SREFP 3 C00063 BC00063  +REFP EC00063
CALL JOB:SEARCH-R1-S13D
SET P054 P006
SFTON3D P054
SMOVL C00064 BC00064 V=166.7  +MOVJ EC00064
SMOVL C00065 BC00065 V=416.7  +MOVJ EC00065
SMOVL C00066 BC00066 V=250.0  +MOVJ EC00066
SREFP 3 C00067 BC00067  +REFP EC00067
CALL JOB:SEARCH-R1-S13D
SET P054 P006
SFTON3D P054
SMOVL C00068 BC00068 V=250.0  +MOVJ EC00068
MOVL C00069 BC00069 V=1000.0  +MOVJ EC00069 VJ=100.00
'EndPath S4207
'Path S4095
SFTOF3D
MOVJ C00070 BC00070 VJ=100.00  +MOVJ EC00070 VJ=100.00
MOVJ C00071 BC00071 VJ=100.00  +MOVJ EC00071 VJ=100.00
SMOVL C00072 BC00072 V=200.0  +MOVJ EC00072
SREFP 3 C00073 BC00073  +REFP EC00073
CALL JOB:SEARCH-R1-S13D
SET P089 P006
SFTON3D P089
SMOVL C00074 BC00074 V=166.7  +MOVJ EC00074
SMOVL C00075 BC00075 V=166.7  +MOVJ EC00075
SREFP 3 C00076 BC00076  +REFP EC00076
CALL JOB:SEARCH-R1-S13D
SET P089 P006
SFTON3D P089
SMOVL C00077 BC00077 V=166.7  +MOVJ EC00077
SMOVL C00078 BC00078 V=166.7  +MOVJ EC00078
SREFP 3 C00079 BC00079  +REFP EC00079
CALL JOB:SEARCH-R1-S13D
SET P089 P006
SFTON3D P089
SMOVL C00080 BC00080 V=166.7  +MOVJ EC00080
SMOVL C00081 BC00081 V=1000.0  +MOVJ EC00081
SFTOF3D
MOVJ C00082 BC00082 VJ=100.00  +MOVJ EC00082 VJ=100.00
MOVL C00083 BC00083 V=666.7  +MOVJ EC00083 VJ=100.00
SMOVL C00084 BC00084 V=166.7  +MOVJ EC00084
SREFP 3 C00085 BC00085  +REFP EC00085
CALL JOB:SEARCH-R1-S13D
SET P034 P006
SFTON3D P034
SMOVL C00086 BC00086 V=250.0  +MOVJ EC00086
SMOVL C00087 BC00087 V=233.3  +MOVJ EC00087
SMOVL C00088 BC00088 V=166.7  +MOVJ EC00088
SREFP 3 C00089 BC00089  +REFP EC00089
CALL JOB:SEARCH-R1-S13D
SET P034 P006
SFTON3D P034
SMOVL C00090 BC00090 V=166.7  +MOVJ EC00090
SMOVL C00091 BC00091 V=166.7  +MOVJ EC00091
SREFP 3 C00092 BC00092  +REFP EC00092
CALL JOB:SEARCH-R1-S13D
SET P034 P006
SFTON3D P034
SMOVL C00093 BC00093 V=166.7  +MOVJ EC00093
MOVJ C00094 BC00094 VJ=50.00  +MOVJ EC00094 VJ=30.00
'EndPath S4095
'Path S4096
SFTOF3D
MOVJ C00095 BC00095 VJ=50.00  +MOVJ EC00095 VJ=30.00
MOVJ C00096 BC00096 VJ=50.00  +MOVJ EC00096 VJ=30.00
MOVJ C00097 BC00097 VJ=50.00  +MOVJ EC00097 VJ=30.00
SMOVL C00098 BC00098 V=166.7  +MOVJ EC00098
SREFP 3 C00099 BC00099  +REFP EC00099
CALL JOB:SEARCH-R1-S13D
SET P061 P006
SFTON3D P061
SMOVL C00100 BC00100 V=166.7  +MOVJ EC00100
SREFP 3 C00101 BC00101  +REFP EC00101
CALL JOB:SEARCH-R1-S13D
SET P061 P006
SFTON3D P061
SMOVL C00102 BC00102 V=166.7  +MOVJ EC00102
SFTOF3D
SMOVL C00103 BC00103 V=666.7  +MOVJ EC00103
SMOVL C00104 BC00104 V=166.7  +MOVJ EC00104
SREFP 3 C00105 BC00105  +REFP EC00105
CALL JOB:SEARCH-R1-S13D
SET P062 P006
SFTON3D P062
SMOVL C00106 BC00106 V=166.7  +MOVJ EC00106
SREFP 3 C00107 BC00107  +REFP EC00107
CALL JOB:SEARCH-R1-S13D
SET P062 P006
SFTON3D P062
SMOVL C00108 BC00108 V=250.0  +MOVJ EC00108
SFTOF3D
SMOVL C00109 BC00109 V=500.0  +MOVJ EC00109
SMOVL C00110 BC00110 V=166.7  +MOVJ EC00110
SREFP 3 C00111 BC00111  +REFP EC00111
CALL JOB:SEARCH-R1-S13D
SET P063 P006
SFTON3D P063
SMOVL C00112 BC00112 V=166.7  +MOVJ EC00112
SREFP 3 C00113 BC00113  +REFP EC00113
CALL JOB:SEARCH-R1-S13D
SET P063 P006
SFTON3D P063
SMOVL C00114 BC00114 V=166.7  +MOVJ EC00114
SFTOF3D
SMOVL C00115 BC00115 V=1000.0  +MOVJ EC00115
MOVJ C00116 BC00116 VJ=100.00  +MOVJ EC00116 VJ=30.00
MOVJ C00117 BC00117 VJ=50.00  +MOVJ EC00117 VJ=30.00
MOVJ C00118 BC00118 VJ=100.00  +MOVJ EC00118 VJ=100.00
MOVL C00119 BC00119 V=666.7  +MOVJ EC00119 VJ=100.00
SMOVL C00120 BC00120 V=166.7  +MOVJ EC00120
SREFP 3 C00121 BC00121  +REFP EC00121
CALL JOB:SEARCH-R1-S13D
SET P023 P006
SFTON3D P023
SMOVL C00122 BC00122 V=166.7  +MOVJ EC00122
SMOVL C00123 BC00123 V=333.3  +MOVJ EC00123
SMOVL C00124 BC00124 V=166.7  +MOVJ EC00124
SREFP 3 C00125 BC00125  +REFP EC00125
CALL JOB:SEARCH-R1-S13D
SET P023 P006
SFTON3D P023
SMOVL C00126 BC00126 V=166.7  +MOVJ EC00126
SMOVL C00127 BC00127 V=166.7  +MOVJ EC00127
SREFP 3 C00128 BC00128  +REFP EC00128
CALL JOB:SEARCH-R1-S13D
SET P023 P006
SFTON3D P023
SMOVL C00129 BC00129 V=166.7  +MOVJ EC00129
MOVL C00130 BC00130 V=1000.0  +MOVJ EC00130 VJ=100.00
'EndPath S4096
MOVJ C00131 BC00131 VJ=100.00  +MOVJ EC00131 VJ=100.00
'Path S4097
SFTOF3D
MOVJ C00132 BC00132 VJ=100.00  +MOVJ EC00132 VJ=100.00
MOVL C00133 BC00133 V=666.7  +MOVJ EC00133 VJ=100.00
SMOVL C00134 BC00134 V=166.7  +MOVJ EC00134
SREFP 3 C00135 BC00135  +REFP EC00135
CALL JOB:SEARCH-R1-S13D
SET P024 P006
SFTON3D P024
SMOVL C00136 BC00136 V=166.7  +MOVJ EC00136
SREFP 3 C00137 BC00137  +REFP EC00137
CALL JOB:SEARCH-R1-S13D
SET P024 P006
SFTON3D P024
SMOVL C00138 BC00138 V=166.7  +MOVJ EC00138
SMOVL C00139 BC00139 V=166.7  +MOVJ EC00139
SREFP 3 C00140 BC00140  +REFP EC00140
CALL JOB:SEARCH-R1-S13D
SET P024 P006
SFTON3D P024
SMOVL C00141 BC00141 V=166.7  +MOVJ EC00141
MOVL C00142 BC00142 V=1000.0  +MOVJ EC00142 VJ=100.00
'EndPath S4097
'Path S4098
SFTOF3D
MOVJ C00143 BC00143 VJ=100.00  +MOVJ EC00143 VJ=100.00
MOVL C00144 BC00144 V=666.7  +MOVJ EC00144 VJ=100.00
SMOVL C00145 BC00145 V=166.7  +MOVJ EC00145
SREFP 3 C00146 BC00146  +REFP EC00146
CALL JOB:SEARCH-R1-S13D
SET P035 P006
SFTON3D P035
SMOVL C00147 BC00147 V=166.7  +MOVJ EC00147
SREFP 3 C00148 BC00148  +REFP EC00148
CALL JOB:SEARCH-R1-S13D
SET P035 P006
SFTON3D P035
SMOVL C00149 BC00149 V=166.7  +MOVJ EC00149
SMOVL C00150 BC00150 V=166.7  +MOVJ EC00150
SMOVL C00151 BC00151 V=166.7  +MOVJ EC00151
SREFP 3 C00152 BC00152  +REFP EC00152
CALL JOB:SEARCH-R1-S13D
SET P035 P006
SFTON3D P035
SMOVL C00153 BC00153 V=166.7  +MOVJ EC00153
MOVL C00154 BC00154 V=1000.0  +MOVJ EC00154 VJ=100.00
'EndPath S4098
'Path S4099
SFTOF3D
MOVJ C00155 BC00155 VJ=100.00  +MOVJ EC00155 VJ=100.00
MOVL C00156 BC00156 V=666.7  +MOVJ EC00156 VJ=100.00
SMOVL C00157 BC00157 V=166.7  +MOVJ EC00157
SREFP 3 C00158 BC00158  +REFP EC00158
CALL JOB:SEARCH-R1-S13D
SET P029 P006
SFTON3D P029
SMOVL C00159 BC00159 V=166.7  +MOVJ EC00159
SREFP 3 C00160 BC00160  +REFP EC00160
CALL JOB:SEARCH-R1-S13D
SET P029 P006
SFTON3D P029
SMOVL C00161 BC00161 V=166.7  +MOVJ EC00161
SMOVL C00162 BC00162 V=250.0  +MOVJ EC00162
SMOVL C00163 BC00163 V=166.7  +MOVJ EC00163
SREFP 3 C00164 BC00164  +REFP EC00164
CALL JOB:SEARCH-R1-S13D
SET P029 P006
SFTON3D P029
SMOVL C00165 BC00165 V=166.7  +MOVJ EC00165
'EndPath S4099
'Path S4855
SFTOF3D
MOVL C00166 BC00166 V=666.7  +MOVJ EC00166 VJ=100.00
SMOVL C00167 BC00167 V=166.7  +MOVJ EC00167
SREFP 3 C00168 BC00168  +REFP EC00168
CALL JOB:SEARCH-R1-S13D
SET P071 P006
SFTON3D P071
SMOVL C00169 BC00169 V=166.7  +MOVJ EC00169
SREFP 3 C00170 BC00170  +REFP EC00170
CALL JOB:SEARCH-R1-S13D
SET P071 P006
SFTON3D P071
SMOVL C00171 BC00171 V=166.7  +MOVJ EC00171
SMOVL C00172 BC00172 V=166.7  +MOVJ EC00172
SREFP 3 C00173 BC00173  +REFP EC00173
CALL JOB:SEARCH-R1-S13D
SET P071 P006
SFTON3D P071
SMOVL C00174 BC00174 V=166.7  +MOVJ EC00174
MOVL C00175 BC00175 V=1000.0  +MOVJ EC00175 VJ=100.00
'EndPath S4855
'Path S4856
SFTOF3D
MOVJ C00176 BC00176 VJ=100.00  +MOVJ EC00176 VJ=100.00
MOVL C00177 BC00177 V=666.7  +MOVJ EC00177 VJ=100.00
SMOVL C00178 BC00178 V=166.7  +MOVJ EC00178
SREFP 3 C00179 BC00179  +REFP EC00179
CALL JOB:SEARCH-R1-S13D
SET P072 P006
SFTON3D P072
SMOVL C00180 BC00180 V=166.7  +MOVJ EC00180
SREFP 3 C00181 BC00181  +REFP EC00181
CALL JOB:SEARCH-R1-S13D
SET P072 P006
SFTON3D P072
SMOVL C00182 BC00182 V=166.7  +MOVJ EC00182
MOVL C00183 BC00183 V=1000.0  +MOVJ EC00183 VJ=100.00
'EndPath S4856
MOVJ C00184 BC00184 VJ=100.00  +MOVJ EC00184 VJ=100.00
'Path S4857
SFTOF3D
MOVJ C00185 BC00185 VJ=100.00  +MOVJ EC00185 VJ=100.00
MOVL C00186 BC00186 V=666.7  +MOVJ EC00186 VJ=100.00
SMOVL C00187 BC00187 V=166.7  +MOVJ EC00187
SREFP 3 C00188 BC00188  +REFP EC00188
CALL JOB:SEARCH-R1-S13D
SET P073 P006
SFTON3D P073
SMOVL C00189 BC00189 V=166.7  +MOVJ EC00189
SMOVL C00190 BC00190 V=166.7  +MOVJ EC00190
SREFP 3 C00191 BC00191  +REFP EC00191
CALL JOB:SEARCH-R1-S13D
SET P073 P006
SFTON3D P073
SMOVL C00192 BC00192 V=166.7  +MOVJ EC00192
SMOVL C00193 BC00193 V=166.7  +MOVJ EC00193
SREFP 3 C00194 BC00194  +REFP EC00194
CALL JOB:SEARCH-R1-S13D
SET P073 P006
SFTON3D P073
SMOVL C00195 BC00195 V=166.7  +MOVJ EC00195
MOVL C00196 BC00196 V=1000.0  +MOVJ EC00196 VJ=100.00
'EndPath S4857
MOVJ C00197 BC00197 VJ=100.00  +MOVJ EC00197 VJ=100.00
'Path S4858
SFTOF3D
MOVJ C00198 BC00198 VJ=100.00  +MOVJ EC00198 VJ=100.00
MOVL C00199 BC00199 V=666.7  +MOVJ EC00199 VJ=100.00
SMOVL C00200 BC00200 V=166.7  +MOVJ EC00200
SREFP 3 C00201 BC00201  +REFP EC00201
CALL JOB:SEARCH-R1-S13D
SET P074 P006
SFTON3D P074
SMOVL C00202 BC00202 V=166.7  +MOVJ EC00202
SREFP 3 C00203 BC00203  +REFP EC00203
CALL JOB:SEARCH-R1-S13D
SET P074 P006
SFTON3D P074
SMOVL C00204 BC00204 V=166.7  +MOVJ EC00204
MOVL C00205 BC00205 V=1000.0  +MOVJ EC00205 VJ=100.00
'EndPath S4858
MOVJ C00206 BC00206 VJ=100.00  +MOVJ EC00206 VJ=100.00
MOVJ C00207 BC00207 VJ=100.00  +MOVJ EC00207 VJ=100.00
'Path S4100
SFTOF3D
MOVJ C00208 BC00208 VJ=100.00  +MOVJ EC00208 VJ=100.00
MOVL C00209 BC00209 V=666.7  +MOVJ EC00209 VJ=100.00
SMOVL C00210 BC00210 V=166.7  +MOVJ EC00210
SREFP 3 C00211 BC00211  +REFP EC00211
CALL JOB:SEARCH-R1-S13D
SET P026 P006
SFTON3D P026
SMOVL C00212 BC00212 V=166.7  +MOVJ EC00212
SREFP 3 C00213 BC00213  +REFP EC00213
CALL JOB:SEARCH-R1-S13D
SET P026 P006
SFTON3D P026
SMOVL C00214 BC00214 V=166.7  +MOVJ EC00214
SMOVL C00215 BC00215 V=666.7  +MOVJ EC00215
SMOVL C00216 BC00216 V=666.7  +MOVJ EC00216
SMOVL C00217 BC00217 V=666.7  +MOVJ EC00217
SMOVL C00218 BC00218 V=166.7  +MOVJ EC00218
SREFP 3 C00219 BC00219  +REFP EC00219
CALL JOB:SEARCH-R1-S13D
SET P026 P006
SFTON3D P026
SMOVL C00220 BC00220 V=250.0  +MOVJ EC00220
SMOVL C00221 BC00221 V=666.7  +MOVJ EC00221
MOVL C00222 BC00222 V=1000.0  +MOVJ EC00222 VJ=100.00
'EndPath S4100
MOVJ C00223 BC00223 VJ=50.00  +MOVJ EC00223 VJ=100.00
'Path S4101
SFTOF3D
MOVJ C00224 BC00224 VJ=50.00  +MOVJ EC00224 VJ=100.00
MOVL C00225 BC00225 V=666.7  +MOVJ EC00225 VJ=100.00
SMOVL C00226 BC00226 V=166.7  +MOVJ EC00226
SREFP 3 C00227 BC00227  +REFP EC00227
CALL JOB:SEARCH-R1-S13D
SET P025 P006
SFTON3D P025
SMOVL C00228 BC00228 V=166.7  +MOVJ EC00228
SREFP 3 C00229 BC00229  +REFP EC00229
CALL JOB:SEARCH-R1-S13D
SET P025 P006
SFTON3D P025
SMOVL C00230 BC00230 V=166.7  +MOVJ EC00230
SMOVL C00231 BC00231 V=333.3  +MOVJ EC00231
SMOVL C00232 BC00232 V=166.7  +MOVJ EC00232
SREFP 3 C00233 BC00233  +REFP EC00233
CALL JOB:SEARCH-R1-S13D
SET P025 P006
SFTON3D P025
SMOVL C00234 BC00234 V=166.7  +MOVJ EC00234
MOVL C00235 BC00235 V=1000.0  +MOVJ EC00235 VJ=100.00
'EndPath S4101
MOVJ C00236 BC00236 VJ=100.00  +MOVJ EC00236 VJ=100.00
'Path S4102
SFTOF3D
MOVJ C00237 BC00237 VJ=100.00  +MOVJ EC00237 VJ=100.00
MOVL C00238 BC00238 V=666.7  +MOVJ EC00238 VJ=100.00
SMOVL C00239 BC00239 V=166.7  +MOVJ EC00239
SREFP 3 C00240 BC00240  +REFP EC00240
CALL JOB:SEARCH-R1-S13D
SET P028 P006
SFTON3D P028
SMOVL C00241 BC00241 V=166.7  +MOVJ EC00241
SREFP 3 C00242 BC00242  +REFP EC00242
CALL JOB:SEARCH-R1-S13D
SET P028 P006
SFTON3D P028
SMOVL C00243 BC00243 V=166.7  +MOVJ EC00243
SMOVL C00244 BC00244 V=333.3  +MOVJ EC00244
SMOVL C00245 BC00245 V=166.7  +MOVJ EC00245
SREFP 3 C00246 BC00246  +REFP EC00246
CALL JOB:SEARCH-R1-S13D
SET P028 P006
SFTON3D P028
SMOVL C00247 BC00247 V=166.7  +MOVJ EC00247
MOVL C00248 BC00248 V=1000.0  +MOVJ EC00248 VJ=100.00
'EndPath S4102
MOVJ C00249 BC00249 VJ=100.00  +MOVJ EC00249 VJ=100.00
'Path S4103
SFTOF3D
MOVJ C00250 BC00250 VJ=100.00  +MOVJ EC00250 VJ=100.00
MOVL C00251 BC00251 V=666.7  +MOVJ EC00251 VJ=100.00
SMOVL C00252 BC00252 V=166.7  +MOVJ EC00252
SREFP 3 C00253 BC00253  +REFP EC00253
CALL JOB:SEARCH-R1-S13D
SET P033 P006
SFTON3D P033
SMOVL C00254 BC00254 V=166.7  +MOVJ EC00254
SMOVL C00255 BC00255 V=166.7  +MOVJ EC00255
SREFP 3 C00256 BC00256  +REFP EC00256
CALL JOB:SEARCH-R1-S13D
SET P033 P006
SFTON3D P033
SMOVL C00257 BC00257 V=166.7  +MOVJ EC00257
SMOVL C00258 BC00258 V=166.7  +MOVJ EC00258
SMOVL C00259 BC00259 V=166.7  +MOVJ EC00259
SREFP 3 C00260 BC00260  +REFP EC00260
CALL JOB:SEARCH-R1-S13D
SET P033 P006
SFTON3D P033
SMOVL C00261 BC00261 V=166.7  +MOVJ EC00261
MOVL C00262 BC00262 V=1000.0  +MOVJ EC00262 VJ=100.00
'EndPath S4103
'Path S4104
SFTOF3D
MOVJ C00263 BC00263 VJ=100.00  +MOVJ EC00263 VJ=100.00
MOVL C00264 BC00264 V=666.7  +MOVJ EC00264 VJ=100.00
SMOVL C00265 BC00265 V=166.7  +MOVJ EC00265
SREFP 3 C00266 BC00266  +REFP EC00266
CALL JOB:SEARCH-R1-S13D
SET P027 P006
SFTON3D P027
SMOVL C00267 BC00267 V=250.0  +MOVJ EC00267
SMOVL C00268 BC00268 V=166.7  +MOVJ EC00268
SREFP 3 C00269 BC00269  +REFP EC00269
CALL JOB:SEARCH-R1-S13D
SET P027 P006
SFTON3D P027
SMOVL C00270 BC00270 V=166.7  +MOVJ EC00270
SMOVL C00271 BC00271 V=166.7  +MOVJ EC00271
SREFP 3 C00272 BC00272  +REFP EC00272
CALL JOB:SEARCH-R1-S13D
SET P027 P006
SFTON3D P027
SMOVL C00273 BC00273 V=166.7  +MOVJ EC00273
MOVL C00274 BC00274 V=1000.0  +MOVJ EC00274 VJ=100.00
'EndPath S4104
MOVJ C00275 BC00275 VJ=100.00  +MOVJ EC00275 VJ=100.00
'Path S4105
SFTOF3D
MOVJ C00276 BC00276 VJ=100.00  +MOVJ EC00276 VJ=100.00
MOVL C00277 BC00277 V=666.7  +MOVJ EC00277 VJ=100.00
SMOVL C00278 BC00278 V=166.7  +MOVJ EC00278
SREFP 3 C00279 BC00279  +REFP EC00279
CALL JOB:SEARCH-R1-S13D
SET P030 P006
SFTON3D P030
SMOVL C00280 BC00280 V=166.7  +MOVJ EC00280
SREFP 3 C00281 BC00281  +REFP EC00281
CALL JOB:SEARCH-R1-S13D
SET P030 P006
SFTON3D P030
SMOVL C00282 BC00282 V=166.7  +MOVJ EC00282
MOVL C00283 BC00283 V=1000.0  +MOVJ EC00283 VJ=100.00
'EndPath S4105
'Path S4106
SFTOF3D
MOVJ C00284 BC00284 VJ=100.00  +MOVJ EC00284 VJ=100.00
MOVL C00285 BC00285 V=666.7  +MOVJ EC00285 VJ=100.00
SMOVL C00286 BC00286 V=166.7  +MOVJ EC00286
SREFP 3 C00287 BC00287  +REFP EC00287
CALL JOB:SEARCH-R1-S13D
SET P031 P006
SFTON3D P031
SMOVL C00288 BC00288 V=166.7  +MOVJ EC00288
SREFP 3 C00289 BC00289  +REFP EC00289
CALL JOB:SEARCH-R1-S13D
SET P031 P006
SFTON3D P031
SMOVL C00290 BC00290 V=166.7  +MOVJ EC00290
MOVL C00291 BC00291 V=1000.0  +MOVJ EC00291 VJ=100.00
'EndPath S4106
MOVJ C00292 BC00292 VJ=100.00  +MOVJ EC00292 VJ=100.00
'Path S4107
SFTOF3D
MOVJ C00293 BC00293 VJ=100.00  +MOVJ EC00293 VJ=100.00
MOVL C00294 BC00294 V=666.7  +MOVJ EC00294 VJ=100.00
SMOVL C00295 BC00295 V=166.7  +MOVJ EC00295
SREFP 3 C00296 BC00296  +REFP EC00296
CALL JOB:SEARCH-R1-S13D
SET P032 P006
SFTON3D P032
SMOVL C00297 BC00297 V=166.7  +MOVJ EC00297
SREFP 3 C00298 BC00298  +REFP EC00298
CALL JOB:SEARCH-R1-S13D
SET P032 P006
SFTON3D P032
SMOVL C00299 BC00299 V=166.7  +MOVJ EC00299
SMOVL C00300 BC00300 V=250.0  +MOVJ EC00300
SMOVL C00301 BC00301 V=166.7  +MOVJ EC00301
SREFP 3 C00302 BC00302  +REFP EC00302
CALL JOB:SEARCH-R1-S13D
SET P032 P006
SFTON3D P032
SMOVL C00303 BC00303 V=166.7  +MOVJ EC00303
MOVL C00304 BC00304 V=1000.0  +MOVJ EC00304 VJ=100.00
'EndPath S4107
'
MOVJ C00305 BC00305 VJ=100.00  +MOVJ EC00305 VJ=100.00
'Path S4208
SFTOF3D
MOVJ C00306 BC00306 VJ=100.00  +MOVJ EC00306 VJ=100.00
MOVL C00307 BC00307 V=666.7  +MOVJ EC00307 VJ=100.00
SMOVL C00308 BC00308 V=166.7  +MOVJ EC00308
SREFP 3 C00309 BC00309  +REFP EC00309
CALL JOB:SEARCH-R1-S13D
SET P052 P006
SFTON3D P052
SMOVL C00310 BC00310 V=166.7  +MOVJ EC00310
SREFP 3 C00311 BC00311  +REFP EC00311
CALL JOB:SEARCH-R1-S13D
SET P052 P006
SFTON3D P052
SMOVL C00312 BC00312 V=166.7  +MOVJ EC00312
SFTOF3D
MOVL C00313 BC00313 V=1000.0  +MOVJ EC00313 VJ=100.00
SMOVL C00314 BC00314 V=500.0  +MOVJ EC00314
SMOVL C00315 BC00315 V=166.7  +MOVJ EC00315
SREFP 3 C00316 BC00316  +REFP EC00316
CALL JOB:SEARCH-R1-S13D
SET P088 P006
SFTON3D P088
SMOVL C00317 BC00317 V=166.7  +MOVJ EC00317
SMOVL C00318 BC00318 V=166.7  +MOVJ EC00318
SMOVL C00319 BC00319 V=166.7  +MOVJ EC00319
SREFP 3 C00320 BC00320  +REFP EC00320
CALL JOB:SEARCH-R1-S13D
SET P088 P006
SFTON3D P088
SMOVL C00321 BC00321 V=333.3  +MOVJ EC00321
SMOVL C00322 BC00322 V=666.7  +MOVJ EC00322
SFTOF3D
'EndPath S4208
MOVJ C00323 BC00323 VJ=100.00  +MOVJ EC00323 VJ=100.00
'Path S4209
SFTOF3D
MOVJ C00324 BC00324 VJ=100.00  +MOVJ EC00324 VJ=100.00
MOVL C00325 BC00325 V=666.7  +MOVJ EC00325 VJ=100.00
SMOVL C00326 BC00326 V=166.7  +MOVJ EC00326
SREFP 3 C00327 BC00327  +REFP EC00327
CALL JOB:SEARCH-R1-S13D
SET P053 P006
SFTON3D P053
SMOVL C00328 BC00328 V=166.7  +MOVJ EC00328
SMOVL C00329 BC00329 V=166.7  +MOVJ EC00329
SREFP 3 C00330 BC00330  +REFP EC00330
CALL JOB:SEARCH-R1-S13D
SET P053 P006
SFTON3D P053
SMOVL C00331 BC00331 V=166.7  +MOVJ EC00331
MOVL C00332 BC00332 V=1000.0  +MOVJ EC00332 VJ=100.00
'EndPath S4209
*BP1
MOVJ C00333 BC00333 VJ=100.00  +MOVJ EC00333 VJ=100.00
'Path W4108
SFTOF3D
SFTON3D P033
MOVJ C00334 BC00334 VJ=100.00  +MOVJ EC00334 VJ=100.00
SMOVL C00335 BC00335 V=666.7  +MOVJ EC00335
SMOVL C00336 BC00336 V=166.7 PL=0  +MOVJ EC00336
MACRO1 MJ#(0) ARGF14
ARCON
SMOVL C00337 BC00337 V=9.2  +MOVJ EC00337
ARCOF
SMOVL C00338 BC00338 V=800.0  +MOVJ EC00338
SMOVL C00339 BC00339 V=1000.0  +MOVJ EC00339
SFTOF3D
'EndPath W4108
'Path W4109
SFTOF3D
MOVJ C00340 BC00340 VJ=100.00  +MOVJ EC00340 VJ=100.00
MOVJ C00341 BC00341 VJ=100.00  +MOVJ EC00341 VJ=100.00
'Path W4110
SFTOF3D
SFTON3D P033
MOVJ C00342 BC00342 VJ=100.00  +MOVJ EC00342 VJ=100.00
SMOVL C00343 BC00343 V=800.0  +MOVJ EC00343
SMOVL C00344 BC00344 V=133.3 PL=0  +MOVJ EC00344
MACRO1 MJ#(0) ARGF9
ARCON
SMOVL C00345 BC00345 V=11.7  +MOVJ EC00345
SMOVL C00346 BC00346 V=11.7  +MOVJ EC00346
SMOVL C00347 BC00347 V=11.7  +MOVJ EC00347
ARCOF
SMOVL C00348 BC00348 V=800.0  +MOVJ EC00348
SMOVL C00349 BC00349 V=1000.0  +MOVJ EC00349
SFTOF3D
'EndPath W4110
MOVJ C00350 BC00350 VJ=100.00  +MOVJ EC00350 VJ=100.00
'9
MOVJ C00351 BC00351 VJ=100.00  +MOVJ EC00351 VJ=100.00
'Path W4111
SFTOF3D
SFTON3D P026
MOVJ C00352 BC00352 VJ=100.00  +MOVJ EC00352 VJ=100.00
SMOVL C00353 BC00353 V=666.7  +MOVJ EC00353
SMOVL C00354 BC00354 V=166.7 PL=0  +MOVJ EC00354
MACRO1 MJ#(0) ARGF14
ARCON
SMOVL C00355 BC00355 V=9.2  +MOVJ EC00355
ARCOF
SMOVL C00356 BC00356 V=800.0  +MOVJ EC00356
SMOVL C00357 BC00357 V=1000.0  +MOVJ EC00357
SFTOF3D
'EndPath W4111
'Path W4112
SFTOF3D
SFTON3D P026
MOVJ C00358 BC00358 VJ=100.00  +MOVJ EC00358 VJ=100.00
SMOVL C00359 BC00359 V=800.0  +MOVJ EC00359
SMOVL C00360 BC00360 V=150.0 PL=0  +MOVJ EC00360
ARCON
SMOVL C00361 BC00361 V=11.7  +MOVJ EC00361
SMOVL C00362 BC00362 V=11.7  +MOVJ EC00362
SMOVL C00363 BC00363 V=11.7  +MOVJ EC00363
ARCOF
SMOVL C00364 BC00364 V=800.0  +MOVJ EC00364
SMOVL C00365 BC00365 V=1000.0  +MOVJ EC00365
SFTOF3D
MOVJ C00366 BC00366 VJ=100.00  +MOVJ EC00366 VJ=100.00
MOVJ C00367 BC00367 VJ=100.00  +MOVJ EC00367 VJ=100.00
'uwaga na podajnik
'Path W4114
SFTOF3D
SFTON3D P026
MOVJ C00368 BC00368 VJ=100.00  +MOVJ EC00368 VJ=100.00
SMOVL C00369 BC00369 V=800.0  +MOVJ EC00369
SMOVL C00370 BC00370 V=150.0 PL=0  +MOVJ EC00370
ARCON
SMOVL C00371 BC00371 V=11.7  +MOVJ EC00371
ARCOF
SMOVL C00372 BC00372 V=800.0  +MOVJ EC00372
SMOVL C00373 BC00373 V=1000.0  +MOVJ EC00373
SFTOF3D
'EndPath W4114
'brak dostepu offset drutu 1cm
'Path W4115
SFTOF3D
SFTON3D P026
MOVJ C00374 BC00374 VJ=100.00  +MOVJ EC00374 VJ=100.00
SMOVL C00375 BC00375 V=800.0  +MOVJ EC00375
SMOVL C00376 BC00376 V=150.0 PL=0  +MOVJ EC00376
ARCON
SMOVL C00377 BC00377 V=11.7  +MOVJ EC00377
ARCOF
SMOVL C00378 BC00378 V=800.0  +MOVJ EC00378
SMOVL C00379 BC00379 V=1000.0  +MOVJ EC00379
SFTOF3D
'EndPath W4115
MOVJ C00380 BC00380 VJ=100.00  +MOVJ EC00380 VJ=100.00
'10
'11
MOVJ C00381 BC00381 VJ=100.00  +MOVJ EC00381 VJ=100.00
'Path W4118
SFTOF3D
SFTON3D P025
MOVJ C00382 BC00382 VJ=100.00  +MOVJ EC00382 VJ=100.00
SMOVL C00383 BC00383 V=800.0  +MOVJ EC00383
SMOVL C00384 BC00384 V=166.7  +MOVJ EC00384
ARCON
SMOVL C00385 BC00385 V=9.2  +MOVJ EC00385
SMOVL C00386 BC00386 V=9.2  +MOVJ EC00386
SMOVL C00387 BC00387 V=9.2  +MOVJ EC00387
SMOVL C00388 BC00388 V=9.2  +MOVJ EC00388
SMOVL C00389 BC00389 V=9.2  +MOVJ EC00389
ARCOF
SMOVL C00390 BC00390 V=800.0  +MOVJ EC00390
SMOVL C00391 BC00391 V=1000.0  +MOVJ EC00391
SFTOF3D
'EndPath W4118
'brak dostepu offset drutu 1cm
MOVJ C00392 BC00392 VJ=100.00  +MOVJ EC00392 VJ=100.00
'Path W4117
SFTOF3D
SFTON3D P025
MOVJ C00393 BC00393 VJ=100.00  +MOVJ EC00393 VJ=100.00
SMOVL C00394 BC00394 V=800.0  +MOVJ EC00394
SMOVL C00395 BC00395 V=166.7 PL=0  +MOVJ EC00395
ARCON
SMOVL C00396 BC00396 V=10.0  +MOVJ EC00396
ARCOF
SMOVL C00397 BC00397 V=800.0  +MOVJ EC00397
SMOVL C00398 BC00398 V=1000.0  +MOVJ EC00398
SFTOF3D
'EndPath W4117
'12
MOVJ C00399 BC00399 VJ=100.00  +MOVJ EC00399 VJ=100.00
MOVJ C00400 BC00400 VJ=100.00  +MOVJ EC00400 VJ=100.00
'Path W4859
SFTOF3D
SFTON3D P073
MOVJ C00401 BC00401 VJ=100.00  +MOVJ EC00401 VJ=100.00
SMOVL C00402 BC00402 V=800.0  +MOVJ EC00402
SMOVL C00403 BC00403 V=150.0 PL=0  +MOVJ EC00403
ARCON
SMOVL C00404 BC00404 V=8.3  +MOVJ EC00404
SFTON3D P074
SMOVL C00405 BC00405 V=9.2  +MOVJ EC00405
SMOVL C00406 BC00406 V=9.2  +MOVJ EC00406
ARCOF
SMOVL C00407 BC00407 V=800.0  +MOVJ EC00407
SMOVL C00408 BC00408 V=1000.0  +MOVJ EC00408
SFTOF3D
'EndPath W4859
MOVJ C00409 BC00409 VJ=100.00  +MOVJ EC00409 VJ=100.00
MOVJ C00410 BC00410 VJ=100.00  +MOVJ EC00410 VJ=100.00
'Path W4119
SFTOF3D
SFTON3D P034
MOVJ C00411 BC00411 VJ=100.00  +MOVJ EC00411 VJ=100.00
SMOVL C00412 BC00412 V=800.0  +MOVJ EC00412
SMOVL C00413 BC00413 V=150.0 PL=0  +MOVJ EC00413
ARCON
SMOVL C00414 BC00414 V=10.0  +MOVJ EC00414
SMOVL C00415 BC00415 V=10.0  +MOVJ EC00415
SMOVL C00416 BC00416 V=10.0  +MOVJ EC00416
ARCOF
SMOVL C00417 BC00417 V=800.0  +MOVJ EC00417
SMOVL C00418 BC00418 V=1000.0  +MOVJ EC00418
SFTOF3D
'EndPath W4119
'Path W4210
SFTOF3D
SFTON3D P050
MOVJ C00419 BC00419 VJ=100.00  +MOVJ EC00419 VJ=100.00
SMOVL C00420 BC00420 V=800.0  +MOVJ EC00420
SMOVL C00421 BC00421 V=150.0 PL=0  +MOVJ EC00421
ARCON
SMOVL C00422 BC00422 V=11.7  +MOVJ EC00422
ARCOF
SMOVL C00423 BC00423 V=800.0  +MOVJ EC00423
SMOVL C00424 BC00424 V=1000.0  +MOVJ EC00424
SFTOF3D
'EndPath W4210
'Path W4211
SFTOF3D
SFTON3D P034
MOVJ C00425 BC00425 VJ=100.00  +MOVJ EC00425 VJ=100.00
SMOVL C00426 BC00426 V=800.0  +MOVJ EC00426
SMOVL C00427 BC00427 V=166.7 PL=0  +MOVJ EC00427
ARCON
SWVON WEV#(66)
SMOVL C00428 BC00428 V=9.2  +MOVJ EC00428
SMOVL C00429 BC00429 V=9.2  +MOVJ EC00429
SMOVL C00430 BC00430 V=9.2  +MOVJ EC00430
ARCOF
SMOVL C00431 BC00431 V=800.0  +MOVJ EC00431
SMOVL C00432 BC00432 V=1000.0  +MOVJ EC00432
MOVJ C00433 BC00433 VJ=30.00  +MOVJ EC00433 VJ=30.00
MOVJ C00434 BC00434 VJ=30.00  +MOVJ EC00434 VJ=30.00
SFTOF3D
MACRO1 MJ#(0) ARGF6
MOVJ C00435 BC00435 VJ=30.00  +MOVJ EC00435 VJ=30.00
SFTON3D P063
SMOVL C00436 BC00436 V=133.3  +MOVJ EC00436
ARCON
SMOVL C00437 BC00437 V=11.7  +MOVJ EC00437
SMOVL C00438 BC00438 V=11.7  +MOVJ EC00438
SMOVL C00439 BC00439 V=11.7  +MOVJ EC00439
SFTON3D P062
SMOVL C00440 BC00440 V=11.7  +MOVJ EC00440
SMOVL C00441 BC00441 V=11.7  +MOVJ EC00441
SFTON3D P061
SMOVL C00442 BC00442 V=11.0  +MOVJ EC00442
SMOVL C00443 BC00443 V=11.0  +MOVJ EC00443
ARCOF
SMOVL C00444 BC00444 V=250.0  +MOVJ EC00444
SFTOF3D
MOVJ C00445 BC00445 VJ=30.00  +MOVJ EC00445 VJ=30.00
MOVJ C00446 BC00446 VJ=30.00  +MOVJ EC00446 VJ=30.00
'EndPath W4211
'Path W4210
SFTOF3D
SFTON3D P054
MOVJ C00447 BC00447 VJ=100.00  +MOVJ EC00447 VJ=100.00
SMOVL C00448 BC00448 V=800.0  +MOVJ EC00448
SMOVL C00449 BC00449 V=150.0 PL=0  +MOVJ EC00449
MACRO1 MJ#(0) ARGF14
ARCON
SWVON WEV#(67)
SMOVL C00450 BC00450 V=10.0  +MOVJ EC00450
SMOVL C00451 BC00451 V=10.0  +MOVJ EC00451
ARCOF
SWVOF
SMOVL C00452 BC00452 V=800.0  +MOVJ EC00452
SMOVL C00453 BC00453 V=1000.0  +MOVJ EC00453
SFTOF3D
'EndPath W4210
'Path W4121
SFTOF3D
SFTON3D P028
MOVJ C00454 BC00454 VJ=100.00  +MOVJ EC00454 VJ=100.00
SMOVL C00455 BC00455 V=800.0  +MOVJ EC00455
SMOVL C00456 BC00456 V=150.0 PL=0  +MOVJ EC00456
ARCON
SMOVL C00457 BC00457 V=9.2  +MOVJ EC00457
SMOVL C00458 BC00458 V=9.2  +MOVJ EC00458
SMOVL C00459 BC00459 V=9.2  +MOVJ EC00459
ARCOF
SMOVL C00460 BC00460 V=800.0  +MOVJ EC00460
SMOVL C00461 BC00461 V=1000.0  +MOVJ EC00461
SFTOF3D
'EndPath W4121
'brak dostepu offset 5mm
MOVJ C00462 BC00462 VJ=100.00  +MOVJ EC00462 VJ=100.00
'Path W4122
SFTOF3D
SFTON3D P028
MOVJ C00463 BC00463 VJ=100.00  +MOVJ EC00463 VJ=100.00
SMOVL C00464 BC00464 V=800.0  +MOVJ EC00464
SMOVL C00465 BC00465 V=166.7 PL=0  +MOVJ EC00465
ARCON
SMOVL C00466 BC00466 V=11.7  +MOVJ EC00466
ARCOF
SMOVL C00467 BC00467 V=800.0  +MOVJ EC00467
SMOVL C00468 BC00468 V=1000.0  +MOVJ EC00468
SFTOF3D
'EndPath W4122
MOVJ C00469 BC00469 VJ=100.00  +MOVJ EC00469 VJ=100.00
'13
MOVJ C00470 BC00470 VJ=100.00  +MOVJ EC00470 VJ=100.00
'Path W4123
SFTOF3D
SFTON3D P030
MOVJ C00471 BC00471 VJ=100.00  +MOVJ EC00471 VJ=100.00
SMOVL C00472 BC00472 V=800.0  +MOVJ EC00472
SMOVL C00473 BC00473 V=150.0 PL=0  +MOVJ EC00473
MACRO1 MJ#(0) ARGF9
ARCON
SWVON WEV#(10)
SFTON3D P031
SMOVL C00474 BC00474 V=12.5  +MOVJ EC00474
ARCOF
SWVOF
SMOVL C00475 BC00475 V=800.0  +MOVJ EC00475
SMOVL C00476 BC00476 V=1000.0  +MOVJ EC00476
SFTOF3D
'EndPath W4123
'14
'15-brak
'Path W4212
SFTOF3D
SFTON3D P052
MOVJ C00477 BC00477 VJ=100.00  +MOVJ EC00477 VJ=100.00
SMOVL C00478 BC00478 V=800.0  +MOVJ EC00478
SMOVL C00479 BC00479 V=150.0 PL=0  +MOVJ EC00479
ARCON
SMOVL C00480 BC00480 V=10.8  +MOVJ EC00480
SMOVL C00481 BC00481 V=10.8  +MOVJ EC00481
SMOVL C00482 BC00482 V=10.8  +MOVJ EC00482
ARCOF
SMOVL C00483 BC00483 V=800.0  +MOVJ EC00483
MACRO1 MJ#(0) ARGF6
SMOVL C00484 BC00484 V=333.3  +MOVJ EC00484
SFTOF3D
'DODAC SHIFT
SFTON3D P088
SMOVL C00485 BC00485 V=133.3  +MOVJ EC00485
ARCON
SMOVL C00486 BC00486 V=10.8  +MOVJ EC00486
ARCOF
SMOVL C00487 BC00487 V=250.0  +MOVJ EC00487
SMOVL C00488 BC00488 V=1000.0  +MOVJ EC00488
SFTOF3D
'EndPath W4212
'16
'Path W4213
SFTOF3D
SFTON3D P053
MOVJ C00489 BC00489 VJ=100.00  +MOVJ EC00489 VJ=100.00
SMOVL C00490 BC00490 V=800.0  +MOVJ EC00490
SMOVL C00491 BC00491 V=150.0 PL=0  +MOVJ EC00491
MACRO1 MJ#(0) ARGF9
ARCON
SMOVL C00492 BC00492 V=10.8  +MOVJ EC00492
SMOVL C00493 BC00493 V=10.8  +MOVJ EC00493
SMOVL C00494 BC00494 V=10.8  +MOVJ EC00494
ARCOF
SMOVL C00495 BC00495 V=800.0  +MOVJ EC00495
SMOVL C00496 BC00496 V=1000.0  +MOVJ EC00496
SFTOF3D
'EndPath W4213
'Path W4124
SFTOF3D
SFTON3D P029
MOVJ C00497 BC00497 VJ=100.00  +MOVJ EC00497 VJ=100.00
SMOVL C00498 BC00498 V=800.0  +MOVJ EC00498
SMOVL C00499 BC00499 V=166.7 PL=0  +MOVJ EC00499
MACRO1 MJ#(0) ARGF14
ARCON
SMOVL C00500 BC00500 V=10.0  +MOVJ EC00500
SMOVL C00501 BC00501 V=10.0  +MOVJ EC00501
ARCOF
SMOVL C00502 BC00502 V=800.0  +MOVJ EC00502
SMOVL C00503 BC00503 V=1000.0  +MOVJ EC00503
SFTOF3D
'EndPath W4124
MOVJ C00504 BC00504 VJ=100.00  +MOVJ EC00504 VJ=100.00
'Path W4125
SFTOF3D
SFTON3D P029
MOVJ C00505 BC00505 VJ=100.00  +MOVJ EC00505 VJ=100.00
SMOVL C00506 BC00506 V=800.0  +MOVJ EC00506
SMOVL C00507 BC00507 V=150.0 PL=0  +MOVJ EC00507
ARCON
SMOVL C00508 BC00508 V=11.7  +MOVJ EC00508
SMOVL C00509 BC00509 V=11.7  +MOVJ EC00509
SMOVL C00510 BC00510 V=11.7  +MOVJ EC00510
ARCOF
SMOVL C00511 BC00511 V=800.0  +MOVJ EC00511
SMOVL C00512 BC00512 V=1000.0  +MOVJ EC00512
SFTOF3D
'EndPath W4125
MOVJ C00513 BC00513 VJ=100.00  +MOVJ EC00513 VJ=100.00
'Path W4126
SFTOF3D
SFTON3D P029
MOVJ C00514 BC00514 VJ=100.00  +MOVJ EC00514 VJ=100.00
SMOVL C00515 BC00515 V=800.0  +MOVJ EC00515
SMOVL C00516 BC00516 V=166.7 PL=0  +MOVJ EC00516
ARCON
SMOVL C00517 BC00517 V=11.7  +MOVJ EC00517
ARCON
SMOVL C00518 BC00518 V=11.7  +MOVJ EC00518
SMOVL C00519 BC00519 V=11.7  +MOVJ EC00519
ARCOF
SMOVL C00520 BC00520 V=800.0  +MOVJ EC00520
SMOVL C00521 BC00521 V=1000.0  +MOVJ EC00521
SFTOF3D
'EndPath W4126
MOVJ C00522 BC00522 VJ=100.00  +MOVJ EC00522 VJ=100.00
'17
'Path W4127
SFTOF3D
SFTON3D P027
MOVJ C00523 BC00523 VJ=100.00  +MOVJ EC00523 VJ=100.00
SMOVL C00524 BC00524 V=800.0  +MOVJ EC00524
SMOVL C00525 BC00525 V=150.0 PL=0  +MOVJ EC00525
ARCON
SMOVL C00526 BC00526 V=10.0  +MOVJ EC00526
ARCOF
SMOVL C00527 BC00527 V=800.0  +MOVJ EC00527
SMOVL C00528 BC00528 V=1000.0  +MOVJ EC00528
SFTOF3D
'EndPath W4127
'Path W4128
SFTOF3D
SFTON3D P027
MOVJ C00529 BC00529 VJ=100.00  +MOVJ EC00529 VJ=100.00
SMOVL C00530 BC00530 V=800.0  +MOVJ EC00530
SMOVL C00531 BC00531 V=150.0 PL=0  +MOVJ EC00531
ARCON
SMOVL C00532 BC00532 V=11.7  +MOVJ EC00532
ARCOF
SMOVL C00533 BC00533 V=800.0  +MOVJ EC00533
SMOVL C00534 BC00534 V=1000.0  +MOVJ EC00534
SFTOF3D
'EndPath W4128
'Path W4129
SFTOF3D
SFTON3D P027
MOVJ C00535 BC00535 VJ=100.00  +MOVJ EC00535 VJ=100.00
SMOVL C00536 BC00536 V=800.0  +MOVJ EC00536
SMOVL C00537 BC00537 V=150.0 PL=0  +MOVJ EC00537
SMOVL C00538 BC00538 V=16.7  +MOVJ EC00538
ARCOF
SMOVL C00539 BC00539 V=800.0  +MOVJ EC00539
SMOVL C00540 BC00540 V=1000.0  +MOVJ EC00540
SFTOF3D
'EndPath W4129
'18
MOVJ C00541 BC00541 VJ=100.00  +MOVJ EC00541 VJ=100.00
'Path W4130
SFTOF3D
SFTON3D P024
MOVJ C00542 BC00542 VJ=100.00  +MOVJ EC00542 VJ=100.00
SMOVL C00543 BC00543 V=800.0  +MOVJ EC00543
SMOVL C00544 BC00544 V=150.0 PL=0  +MOVJ EC00544
ARCON
SMOVL C00545 BC00545 V=9.2  +MOVJ EC00545
SMOVL C00546 BC00546 V=9.2  +MOVJ EC00546
SMOVL C00547 BC00547 V=9.2  +MOVJ EC00547
SMOVL C00548 BC00548 V=9.2  +MOVJ EC00548
ARCOF
SMOVL C00549 BC00549 V=800.0  +MOVJ EC00549
SMOVL C00550 BC00550 V=1000.0  +MOVJ EC00550
SFTOF3D
'EndPath W4130
'Path W4860
SFTOF3D
SFTON3D P071
MOVJ C00551 BC00551 VJ=100.00  +MOVJ EC00551 VJ=100.00
SMOVL C00552 BC00552 V=800.0  +MOVJ EC00552
SMOVL C00553 BC00553 V=150.0 PL=0  +MOVJ EC00553
MACRO1 MJ#(0) ARGF9
ARCON
SMOVL C00554 BC00554 V=9.2  +MOVJ EC00554
SFTON3D P072
ARCON
SMOVL C00555 BC00555 V=9.2  +MOVJ EC00555
SMOVL C00556 BC00556 V=9.2  +MOVJ EC00556
ARCOF
SMOVL C00557 BC00557 V=800.0  +MOVJ EC00557
SMOVL C00558 BC00558 V=1000.0  +MOVJ EC00558
SFTOF3D
'EndPath W4860
'19
MOVJ C00559 BC00559 VJ=100.00  +MOVJ EC00559 VJ=100.00
'Path W4131
SFTOF3D
SFTON3D P023
MOVJ C00560 BC00560 VJ=100.00  +MOVJ EC00560 VJ=100.00
SMOVL C00561 BC00561 V=800.0  +MOVJ EC00561
SMOVL C00562 BC00562 V=166.7 PL=0  +MOVJ EC00562
MACRO1 MJ#(0) ARGF9
ARCON
SWVON WEV#(60)
SMOVL C00563 BC00563 V=7.5  +MOVJ EC00563
SMOVL C00564 BC00564 V=7.5  +MOVJ EC00564
SMOVL C00565 BC00565 V=7.5  +MOVJ EC00565
ARCOF
SWVOF
SMOVL C00566 BC00566 V=800.0  +MOVJ EC00566
SMOVL C00567 BC00567 V=1000.0  +MOVJ EC00567
SFTOF3D
'EndPath W4131
MOVJ C00568 BC00568 VJ=100.00  +MOVJ EC00568 VJ=100.00
'Path W4214
SFTOF3D
SFTON3D P089
MOVJ C00569 BC00569 VJ=100.00  +MOVJ EC00569 VJ=100.00
SMOVL C00570 BC00570 V=800.0  +MOVJ EC00570
SMOVL C00571 BC00571 V=150.0 PL=0  +MOVJ EC00571
MACRO1 MJ#(0) ARGF9
ARCON
SMOVL C00572 BC00572 V=9.2  +MOVJ EC00572
SFTON3D P050
SMOVL C00573 BC00573 V=9.2  +MOVJ EC00573
SMOVL C00574 BC00574 V=9.2  +MOVJ EC00574
ARCOF
SMOVL C00575 BC00575 V=800.0  +MOVJ EC00575
SMOVL C00576 BC00576 V=1000.0  +MOVJ EC00576
SFTOF3D
'EndPath W4214
'Path W4215
SFTOF3D
SFTON3D P051
MOVJ C00577 BC00577 VJ=100.00  +MOVJ EC00577 VJ=100.00
SMOVL C00578 BC00578 V=800.0  +MOVJ EC00578
SMOVL C00579 BC00579 V=150.0 PL=0  +MOVJ EC00579
MACRO1 MJ#(0) ARGF9
ARCON
SWVON WEV#(60)
SMOVL C00580 BC00580 V=7.5  +MOVJ EC00580
SMOVL C00581 BC00581 V=7.5  +MOVJ EC00581
SMOVL C00582 BC00582 V=7.5  +MOVJ EC00582
ARCOF
SWVOF
SMOVL C00583 BC00583 V=800.0  +MOVJ EC00583
SMOVL C00584 BC00584 V=1000.0  +MOVJ EC00584
SFTOF3D
'EndPath W4215
MOVJ C00585 BC00585 VJ=100.00  +MOVJ EC00585 VJ=100.00
'20
'offset 5mm
MOVJ C00586 BC00586 VJ=100.00  +MOVJ EC00586 VJ=100.00
MOVJ C00587 BC00587 VJ=100.00  +MOVJ EC00587 VJ=100.00
'Path W4132
SFTOF3D
SFTON3D P032
MOVJ C00588 BC00588 VJ=100.00  +MOVJ EC00588 VJ=100.00
SMOVL C00589 BC00589 V=800.0  +MOVJ EC00589
SMOVL C00590 BC00590 V=150.0 PL=0  +MOVJ EC00590
ARCON
SMOVL C00591 BC00591 V=10.0  +MOVJ EC00591
SMOVL C00592 BC00592 V=10.0  +MOVJ EC00592
ARCOF
SMOVL C00593 BC00593 V=800.0  +MOVJ EC00593
SMOVL C00594 BC00594 V=1000.0  +MOVJ EC00594
SFTOF3D
JUMP *FFF
'EndPath W4132
'Path W4133
SFTOF3D
SFTON3D P032
MOVJ C00595 BC00595 VJ=100.00  +MOVJ EC00595 VJ=100.00
SMOVL C00596 BC00596 V=800.0  +MOVJ EC00596
SMOVL C00597 BC00597 V=166.7 PL=0  +MOVJ EC00597
ARCON
SMOVL C00598 BC00598 V=10.0  +MOVJ EC00598
ARCOF
SMOVL C00599 BC00599 V=800.0  +MOVJ EC00599
SMOVL C00600 BC00600 V=1000.0  +MOVJ EC00600
SFTOF3D
'EndPath W4133
'Path W4134
SFTOF3D
SFTON3D P032
MOVJ C00601 BC00601 VJ=100.00  +MOVJ EC00601 VJ=100.00
SMOVL C00602 BC00602 V=800.0  +MOVJ EC00602
SMOVL C00603 BC00603 V=150.0 PL=0  +MOVJ EC00603
ARCON
SMOVL C00604 BC00604 V=10.0  +MOVJ EC00604
ARCOF
SMOVL C00605 BC00605 V=800.0  +MOVJ EC00605
*FFF
SMOVL C00606 BC00606 V=1000.0  +MOVJ EC00606
SFTOF3D
'EndPath W4134
'offset 5mm
MOVJ C00607 BC00607 VJ=100.00  +MOVJ EC00607 VJ=100.00
'Path W4135
SFTOF3D
SFTON3D P032
MOVJ C00608 BC00608 VJ=100.00  +MOVJ EC00608 VJ=100.00
SMOVL C00609 BC00609 V=800.0  +MOVJ EC00609
SMOVL C00610 BC00610 V=166.7 PL=0  +MOVJ EC00610
ARCON
SMOVL C00611 BC00611 V=10.0  +MOVJ EC00611
ARCOF
SMOVL C00612 BC00612 V=800.0  +MOVJ EC00612
SMOVL C00613 BC00613 V=1000.0  +MOVJ EC00613
SFTOF3D
'EndPath W4135
MOVJ C00614 BC00614 VJ=100.00  +MOVJ EC00614 VJ=100.00
'Path W4136
SFTOF3D
SFTON3D P032
MOVJ C00615 BC00615 VJ=100.00  +MOVJ EC00615 VJ=100.00
SMOVL C00616 BC00616 V=800.0  +MOVJ EC00616
SMOVL C00617 BC00617 V=166.7 PL=0  +MOVJ EC00617
ARCON
SMOVL C00618 BC00618 V=11.7  +MOVJ EC00618
SMOVL C00619 BC00619 V=11.7  +MOVJ EC00619
ARCOF
SMOVL C00620 BC00620 V=800.0  +MOVJ EC00620
SMOVL C00621 BC00621 V=1000.0  +MOVJ EC00621
SFTOF3D
'EndPath W4136
MOVJ C00622 BC00622 VJ=100.00  +MOVJ EC00622 VJ=100.00
MOVJ C00623 BC00623 VJ=100.00  +MOVJ EC00623 VJ=100.00
'Path W4137
SFTOF3D
SFTON3D P021
MOVJ C00624 BC00624 VJ=100.00  +MOVJ EC00624 VJ=100.00
SMOVL C00625 BC00625 V=800.0  +MOVJ EC00625
SMOVL C00626 BC00626 V=150.0 PL=0  +MOVJ EC00626
MACRO1 MJ#(0) ARGF9
ARCON
SFTON3D P022
SMOVL C00627 BC00627 V=10.0  +MOVJ EC00627
ARCOF
SMOVL C00628 BC00628 V=800.0  +MOVJ EC00628
SMOVL C00629 BC00629 V=1000.0  +MOVJ EC00629
SFTOF3D
'EndPath W4137
MOVJ C00630 BC00630 VJ=100.00  +MOVJ EC00630 VJ=100.00
'Path W4724
SFTOF3D
SFTON3D P095
MOVJ C00631 BC00631 VJ=100.00  +MOVJ EC00631 VJ=100.00
SMOVL C00632 BC00632 V=800.0  +MOVJ EC00632
SMOVL C00633 BC00633 V=150.0 PL=0  +MOVJ EC00633
ARCON
SMOVL C00634 BC00634 V=10.0  +MOVJ EC00634
SMOVL C00635 BC00635 V=10.0  +MOVJ EC00635
SMOVL C00636 BC00636 V=10.0  +MOVJ EC00636
ARCOF
SMOVL C00637 BC00637 V=800.0  +MOVJ EC00637
SMOVL C00638 BC00638 V=1000.0  +MOVJ EC00638
SFTOF3D
'EndPath W4724
'Path W4725
SFTOF3D
SFTON3D P096
MOVJ C00639 BC00639 VJ=100.00  +MOVJ EC00639 VJ=100.00
SMOVL C00640 BC00640 V=800.0  +MOVJ EC00640
SMOVL C00641 BC00641 V=150.0 PL=0  +MOVJ EC00641
ARCON
SMOVL C00642 BC00642 V=10.0  +MOVJ EC00642
SMOVL C00643 BC00643 V=10.0  +MOVJ EC00643
ARCOF
SMOVL C00644 BC00644 V=800.0  +MOVJ EC00644
SMOVL C00645 BC00645 V=1000.0  +MOVJ EC00645
SFTOF3D
'EndPath W4725
MOVJ C00646 BC00646 VJ=100.00  +MOVJ EC00646 VJ=100.00
'Path W4861
SFTOF3D
SFTON3D P071
MOVJ C00647 BC00647 VJ=100.00  +MOVJ EC00647 VJ=100.00
SMOVL C00648 BC00648 V=800.0  +MOVJ EC00648
SMOVL C00649 BC00649 V=150.0 PL=0  +MOVJ EC00649
MACRO1 MJ#(0) ARGF14
ARCON
SMOVL C00650 BC00650 V=9.2  +MOVJ EC00650
SFTON3D P073
SMOVL C00651 BC00651 V=9.2  +MOVJ EC00651
SMOVL C00652 BC00652 V=9.2  +MOVJ EC00652
ARCOF
SMOVL C00653 BC00653 V=800.0  +MOVJ EC00653
SMOVL C00654 BC00654 V=1000.0  +MOVJ EC00654
SFTOF3D
'EndPath W4861
MOVJ C00655 BC00655 VJ=100.00  +MOVJ EC00655 VJ=100.00
MOVJ C00656 BC00656 VJ=100.00  +MOVJ EC00656 VJ=100.00
CALL JOB:CLEAN-R1_KM_NEW
'cut_wire_dol
'cut_wire_dol
'cut_wire_dol
MOVJ C00657 BC00657 VJ=100.00  +MOVJ EC00657 VJ=100.00
MOVJ C00658 BC00658 VJ=100.00  +MOVJ EC00658 VJ=100.00
MOVJ C00659 BC00659 VJ=100.00  +MOVJ EC00659 VJ=100.00
'Path S4138
SFTOF3D
MOVJ C00660 BC00660 VJ=100.00  +MOVJ EC00660 VJ=100.00
MOVL C00661 BC00661 V=800.0  +MOVJ EC00661 VJ=100.00
SMOVL C00662 BC00662 V=166.7  +MOVJ EC00662
SREFP 3 C00663 BC00663  +REFP EC00663
CALL JOB:SEARCH-R1-S13D
SET P049 P006
SFTON3D P049
SMOVL C00664 BC00664 V=166.7  +MOVJ EC00664
SMOVL C00665 BC00665 V=166.7  +MOVJ EC00665
SREFP 3 C00666 BC00666  +REFP EC00666
CALL JOB:SEARCH-R1-S13D
SET P049 P006
SFTON3D P049
SMOVL C00667 BC00667 V=166.7  +MOVJ EC00667
SMOVL C00668 BC00668 V=166.7  +MOVJ EC00668
SMOVL C00669 BC00669 V=166.7  +MOVJ EC00669
SMOVL C00670 BC00670 V=166.7  +MOVJ EC00670
SREFP 3 C00671 BC00671  +REFP EC00671
CALL JOB:SEARCH-R1-S13D
SET P049 P006
SFTON3D P049
SMOVL C00672 BC00672 V=166.7  +MOVJ EC00672
MOVL C00673 BC00673 V=800.0  +MOVJ EC00673 VJ=100.00
MOVL C00674 BC00674 V=1000.0  +MOVJ EC00674 VJ=100.00
'EndPath S4138
'Path S4139
SFTOF3D
MOVJ C00675 BC00675 VJ=100.00  +MOVJ EC00675 VJ=100.00
MOVL C00676 BC00676 V=800.0  +MOVJ EC00676 VJ=100.00
SMOVL C00677 BC00677 V=166.7  +MOVJ EC00677
SREFP 3 C00678 BC00678  +REFP EC00678
CALL JOB:SEARCH-R1-S13D
SET P048 P006
SFTON3D P048
SMOVL C00679 BC00679 V=166.7  +MOVJ EC00679
SMOVL C00680 BC00680 V=166.7  +MOVJ EC00680
SREFP 3 C00681 BC00681  +REFP EC00681
CALL JOB:SEARCH-R1-S13D
SET P048 P006
SFTON3D P048
SMOVL C00682 BC00682 V=166.7  +MOVJ EC00682
MOVL C00683 BC00683 V=800.0  +MOVJ EC00683 VJ=100.00
MOVL C00684 BC00684 V=1000.0  +MOVJ EC00684 VJ=100.00
'EndPath S4139
'Path S4140
SFTOF3D
MOVJ C00685 BC00685 VJ=100.00  +MOVJ EC00685 VJ=100.00
MOVL C00686 BC00686 V=800.0  +MOVJ EC00686 VJ=100.00
SMOVL C00687 BC00687 V=166.7  +MOVJ EC00687
SREFP 3 C00688 BC00688  +REFP EC00688
CALL JOB:SEARCH-R1-S13D
SET P047 P006
SFTON3D P047
SMOVL C00689 BC00689 V=166.7  +MOVJ EC00689
SMOVL C00690 BC00690 V=166.7  +MOVJ EC00690
SREFP 3 C00691 BC00691  +REFP EC00691
CALL JOB:SEARCH-R1-S13D
SET P047 P006
SFTON3D P047
SMOVL C00692 BC00692 V=166.7  +MOVJ EC00692
MOVL C00693 BC00693 V=800.0  +MOVJ EC00693 VJ=100.00
MOVL C00694 BC00694 V=1000.0  +MOVJ EC00694 VJ=100.00
'EndPath S4140
MOVJ C00695 BC00695 VJ=100.00  +MOVJ EC00695 VJ=100.00
MOVJ C00696 BC00696 VJ=100.00  +MOVJ EC00696 VJ=100.00
MOVJ C00697 BC00697 VJ=100.00  +MOVJ EC00697 VJ=100.00
MOVJ C00698 BC00698 VJ=100.00  +MOVJ EC00698 VJ=100.00
'Path S4141
SFTOF3D
MOVJ C00699 BC00699 VJ=100.00  +MOVJ EC00699 VJ=100.00
MOVL C00700 BC00700 V=800.0  +MOVJ EC00700 VJ=100.00
SMOVL C00701 BC00701 V=166.7  +MOVJ EC00701
SREFP 3 C00702 BC00702  +REFP EC00702
CALL JOB:SEARCH-R1-S13D
SET P046 P006
SFTON3D P046
SMOVL C00703 BC00703 V=166.7  +MOVJ EC00703
SMOVL C00704 BC00704 V=166.7  +MOVJ EC00704
SREFP 3 C00705 BC00705  +REFP EC00705
CALL JOB:SEARCH-R1-S13D
SET P046 P006
SFTON3D P046
SMOVL C00706 BC00706 V=166.7  +MOVJ EC00706
MOVL C00707 BC00707 V=1000.0  +MOVJ EC00707 VJ=100.00
'EndPath S4141
'Path S4142
SFTOF3D
MOVJ C00708 BC00708 VJ=100.00  +MOVJ EC00708 VJ=100.00
MOVL C00709 BC00709 V=800.0  +MOVJ EC00709 VJ=100.00
SMOVL C00710 BC00710 V=166.7  +MOVJ EC00710
SREFP 3 C00711 BC00711  +REFP EC00711
CALL JOB:SEARCH-R1-S13D
SET P045 P006
SFTON3D P045
SMOVL C00712 BC00712 V=166.7  +MOVJ EC00712
SMOVL C00713 BC00713 V=166.7  +MOVJ EC00713
SREFP 3 C00714 BC00714  +REFP EC00714
CALL JOB:SEARCH-R1-S13D
SET P045 P006
SFTON3D P045
SMOVL C00715 BC00715 V=166.7  +MOVJ EC00715
MOVL C00716 BC00716 V=1000.0  +MOVJ EC00716 VJ=100.00
'EndPath S4142
'Path S4143
SFTOF3D
MOVJ C00717 BC00717 VJ=100.00  +MOVJ EC00717 VJ=100.00
MOVL C00718 BC00718 V=800.0  +MOVJ EC00718 VJ=100.00
SMOVL C00719 BC00719 V=166.7  +MOVJ EC00719
SREFP 3 C00720 BC00720  +REFP EC00720
CALL JOB:SEARCH-R1-S13D
SET P044 P006
SFTON3D P044
SMOVL C00721 BC00721 V=166.7  +MOVJ EC00721
SMOVL C00722 BC00722 V=166.7  +MOVJ EC00722
SREFP 3 C00723 BC00723  +REFP EC00723
CALL JOB:SEARCH-R1-S13D
SET P044 P006
SFTON3D P044
SMOVL C00724 BC00724 V=166.7  +MOVJ EC00724
MOVL C00725 BC00725 V=1000.0  +MOVJ EC00725 VJ=100.00
'EndPath S4143
MOVJ C00726 BC00726 VJ=100.00  +MOVJ EC00726 VJ=100.00
MOVJ C00727 BC00727 VJ=100.00  +MOVJ EC00727 VJ=100.00
'Path S4144
SFTOF3D
MOVJ C00728 BC00728 VJ=100.00  +MOVJ EC00728 VJ=100.00
MOVL C00729 BC00729 V=800.0  +MOVJ EC00729 VJ=100.00
SMOVL C00730 BC00730 V=166.7  +MOVJ EC00730
SREFP 3 C00731 BC00731  +REFP EC00731
CALL JOB:SEARCH-R1-S13D
SET P043 P006
SFTON3D P043
SMOVL C00732 BC00732 V=166.7  +MOVJ EC00732
SMOVL C00733 BC00733 V=166.7  +MOVJ EC00733
SREFP 3 C00734 BC00734  +REFP EC00734
CALL JOB:SEARCH-R1-S13D
SET P043 P006
SFTON3D P043
SMOVL C00735 BC00735 V=166.7  +MOVJ EC00735
MOVL C00736 BC00736 V=1000.0  +MOVJ EC00736 VJ=100.00
'EndPath S4144
'Path S4145
SFTOF3D
MOVJ C00737 BC00737 VJ=100.00  +MOVJ EC00737 VJ=100.00
MOVL C00738 BC00738 V=800.0  +MOVJ EC00738 VJ=100.00
SMOVL C00739 BC00739 V=166.7  +MOVJ EC00739
SREFP 3 C00740 BC00740  +REFP EC00740
CALL JOB:SEARCH-R1-S13D
SET P042 P006
SFTON3D P042
SMOVL C00741 BC00741 V=166.7  +MOVJ EC00741
SMOVL C00742 BC00742 V=166.7  +MOVJ EC00742
SREFP 3 C00743 BC00743  +REFP EC00743
CALL JOB:SEARCH-R1-S13D
SET P042 P006
SFTON3D P042
SMOVL C00744 BC00744 V=166.7  +MOVJ EC00744
MOVL C00745 BC00745 V=1000.0  +MOVJ EC00745 VJ=100.00
'EndPath S4145
'Path S4146
SFTOF3D
MOVJ C00746 BC00746 VJ=100.00  +MOVJ EC00746 VJ=100.00
MOVL C00747 BC00747 V=666.7  +MOVJ EC00747 VJ=100.00
SMOVL C00748 BC00748 V=166.7  +MOVJ EC00748
SREFP 3 C00749 BC00749  +REFP EC00749
CALL JOB:SEARCH-R1-S13D
SET P041 P006
SFTON3D P041
SMOVL C00750 BC00750 V=250.0  +MOVJ EC00750
SMOVL C00751 BC00751 V=166.7  +MOVJ EC00751
SREFP 3 C00752 BC00752  +REFP EC00752
CALL JOB:SEARCH-R1-S13D
SET P041 P006
SFTON3D P041
SMOVL C00753 BC00753 V=166.7  +MOVJ EC00753
SMOVL C00754 BC00754 V=166.7  +MOVJ EC00754
SREFP 3 C00755 BC00755  +REFP EC00755
CALL JOB:SEARCH-R1-S13D
SET P041 P006
SFTON3D P041
SMOVL C00756 BC00756 V=166.7  +MOVJ EC00756
MOVL C00757 BC00757 V=1000.0  +MOVJ EC00757 VJ=100.00
'EndPath S4146
'Path S4147
SFTOF3D
MOVJ C00758 BC00758 VJ=100.00  +MOVJ EC00758 VJ=100.00
SMOVL C00759 BC00759 V=666.7  +MOVJ EC00759
SMOVL C00760 BC00760 V=166.7  +MOVJ EC00760
SREFP 3 C00761 BC00761  +REFP EC00761
CALL JOB:SEARCH-R1-S13D
SET P040 P006
SFTON3D P040
SMOVL C00762 BC00762 V=166.7  +MOVJ EC00762
SMOVL C00763 BC00763 V=800.0  +MOVJ EC00763
SMOVL C00764 BC00764 V=166.7  +MOVJ EC00764
SREFP 3 C00765 BC00765  +REFP EC00765
CALL JOB:SEARCH-R1-S13D
SET P040 P006
SFTON3D P040
SMOVL C00766 BC00766 V=166.7  +MOVJ EC00766
SMOVL C00767 BC00767 V=166.7  +MOVJ EC00767
SREFP 3 C00768 BC00768  +REFP EC00768
CALL JOB:SEARCH-R1-S13D
SET P040 P006
SFTON3D P040
SMOVL C00769 BC00769 V=166.7  +MOVJ EC00769
MOVL C00770 BC00770 V=1000.0  +MOVJ EC00770 VJ=100.00
'EndPath S4147
'Path W4148
SFTOF3D
SFTON3D P040
MOVJ C00771 BC00771 VJ=100.00  +MOVJ EC00771 VJ=100.00
SMOVL C00772 BC00772 V=800.0  +MOVJ EC00772
SMOVL C00773 BC00773 V=150.0 PL=0  +MOVJ EC00773
ARCON
SMOVL C00774 BC00774 V=10.0  +MOVJ EC00774
ARCOF
SMOVL C00775 BC00775 V=800.0  +MOVJ EC00775
SMOVL C00776 BC00776 V=1000.0  +MOVJ EC00776
SFTOF3D
'EndPath W4148
'Path W4149
SFTOF3D
SFTON3D P040
MOVJ C00777 BC00777 VJ=100.00  +MOVJ EC00777 VJ=100.00
SMOVL C00778 BC00778 V=800.0  +MOVJ EC00778
SMOVL C00779 BC00779 V=150.0 PL=0  +MOVJ EC00779
ARCON
SMOVL C00780 BC00780 V=11.7  +MOVJ EC00780
ARCOF
SMOVL C00781 BC00781 V=800.0  +MOVJ EC00781
SMOVL C00782 BC00782 V=1000.0  +MOVJ EC00782
SFTOF3D
'EndPath W4149
'Path W4150
SFTOF3D
SFTON3D P040
MOVJ C00783 BC00783 VJ=15.00  +MOVJ EC00783 VJ=15.00
MOVJ C00784 BC00784 VJ=100.00  +MOVJ EC00784 VJ=100.00
SMOVL C00785 BC00785 V=800.0  +MOVJ EC00785
SMOVL C00786 BC00786 V=150.0 PL=0  +MOVJ EC00786
ARCON
SMOVL C00787 BC00787 V=11.7  +MOVJ EC00787
ARCOF
SMOVL C00788 BC00788 V=800.0  +MOVJ EC00788
SMOVL C00789 BC00789 V=1000.0  +MOVJ EC00789
SFTOF3D
'EndPath W4150
'
MOVJ C00790 BC00790 VJ=100.00  +MOVJ EC00790 VJ=100.00
MOVJ C00791 BC00791 VJ=100.00  +MOVJ EC00791 VJ=100.00
'Path W4151
SFTOF3D
SFTON3D P045
MOVJ C00792 BC00792 VJ=100.00  +MOVJ EC00792 VJ=100.00
SMOVL C00793 BC00793 V=800.0  +MOVJ EC00793
SMOVL C00794 BC00794 V=150.0 PL=0  +MOVJ EC00794
MACRO1 MJ#(0) ARGF9
ARCON
SMOVL C00795 BC00795 V=11.7  +MOVJ EC00795
ARCOF
SMOVL C00796 BC00796 V=800.0  +MOVJ EC00796
SMOVL C00797 BC00797 V=1000.0  +MOVJ EC00797
SFTOF3D
'EndPath W4151
'Path W4152
SFTOF3D
SFTON3D P044
MOVJ C00798 BC00798 VJ=100.00  +MOVJ EC00798 VJ=100.00
SMOVL C00799 BC00799 V=800.0  +MOVJ EC00799
SMOVL C00800 BC00800 V=166.7 PL=0  +MOVJ EC00800
ARCON
SMOVL C00801 BC00801 V=11.7  +MOVJ EC00801
ARCOF
SMOVL C00802 BC00802 V=800.0  +MOVJ EC00802
SMOVL C00803 BC00803 V=1000.0  +MOVJ EC00803
SFTOF3D
'EndPath W4152
'Path W4153
SFTOF3D
SFTON3D P046
MOVJ C00804 BC00804 VJ=100.00  +MOVJ EC00804 VJ=100.00
SMOVL C00805 BC00805 V=800.0  +MOVJ EC00805
SMOVL C00806 BC00806 V=166.7 PL=0  +MOVJ EC00806
MACRO1 MJ#(0) ARGF14
ARCON
SMOVL C00807 BC00807 V=10.0  +MOVJ EC00807
SMOVL C00808 BC00808 V=10.0  +MOVJ EC00808
ARCOF
SMOVL C00809 BC00809 V=800.0  +MOVJ EC00809
SMOVL C00810 BC00810 V=1000.0  +MOVJ EC00810
SFTOF3D
'EndPath W4153
MOVJ C00811 BC00811 VJ=100.00  +MOVJ EC00811 VJ=100.00
MOVJ C00812 BC00812 VJ=100.00  +MOVJ EC00812 VJ=100.00
MOVJ C00813 BC00813 VJ=100.00  +MOVJ EC00813 VJ=100.00
MOVJ C00814 BC00814 VJ=100.00  +MOVJ EC00814 VJ=100.00
'1
'uwaga na podajnik
'Path W4154
SFTOF3D
SFTON3D P048
MOVJ C00815 BC00815 VJ=100.00  +MOVJ EC00815 VJ=100.00
SMOVL C00816 BC00816 V=800.0  +MOVJ EC00816
SMOVL C00817 BC00817 V=150.0 PL=0  +MOVJ EC00817
ARCON
SMOVL C00818 BC00818 V=10.0  +MOVJ EC00818
ARCOF
SMOVL C00819 BC00819 V=800.0  +MOVJ EC00819
SMOVL C00820 BC00820 V=1000.0  +MOVJ EC00820
SFTOF3D
'EndPath W4154
'Path W4155
SFTOF3D
SFTON3D P049
MOVJ C00821 BC00821 VJ=100.00  +MOVJ EC00821 VJ=100.00
SMOVL C00822 BC00822 V=800.0  +MOVJ EC00822
SMOVL C00823 BC00823 V=150.0 PL=0  +MOVJ EC00823
MACRO1 MJ#(0) ARGF6
ARCON
SMOVL C00824 BC00824 V=9.2  +MOVJ EC00824
SMOVL C00825 BC00825 V=9.2  +MOVJ EC00825
SMOVL C00826 BC00826 V=9.2  +MOVJ EC00826
SMOVL C00827 BC00827 V=9.2  +MOVJ EC00827
SMOVL C00828 BC00828 V=9.2  +MOVJ EC00828
ARCOF
SMOVL C00829 BC00829 V=800.0  +MOVJ EC00829
SMOVL C00830 BC00830 V=500.0  +MOVJ EC00830
SMOVL C00831 BC00831 V=133.3  +MOVJ EC00831
ARCON
SMOVL C00832 BC00832 V=13.3  +MOVJ EC00832
ARCOF
SMOVL C00833 BC00833 V=166.7  +MOVJ EC00833
ARCON
SMOVL C00834 BC00834 V=10.0  +MOVJ EC00834
ARCOF
SMOVL C00835 BC00835 V=250.0  +MOVJ EC00835
SMOVL C00836 BC00836 V=500.0  +MOVJ EC00836
SMOVL C00837 BC00837 V=500.0  +MOVJ EC00837
SMOVL C00838 BC00838 V=500.0  +MOVJ EC00838
SMOVL C00839 BC00839 V=133.3  +MOVJ EC00839
ARCON
SMOVL C00840 BC00840 V=13.3  +MOVJ EC00840
ARCOF
SMOVL C00841 BC00841 V=166.7  +MOVJ EC00841
SMOVL C00842 BC00842 V=166.7  +MOVJ EC00842
ARCON
SMOVL C00843 BC00843 V=10.0  +MOVJ EC00843
ARCOF
SMOVL C00844 BC00844 V=800.0  +MOVJ EC00844
SFTOF3D
'EndPath W4155
MOVJ C00845 BC00845 VJ=100.00  +MOVJ EC00845 VJ=100.00
MOVJ C00846 BC00846 VJ=100.00  +MOVJ EC00846 VJ=100.00
MOVJ C00847 BC00847 VJ=100.00  +MOVJ EC00847 VJ=100.00
MOVJ C00848 BC00848 VJ=100.00  +MOVJ EC00848 VJ=100.00
'2
'Path W4156
SFTOF3D
SFTON3D P043
MOVJ C00849 BC00849 VJ=100.00  +MOVJ EC00849 VJ=100.00
SMOVL C00850 BC00850 V=800.0  +MOVJ EC00850
SMOVL C00851 BC00851 V=166.7 PL=0  +MOVJ EC00851
MACRO1 MJ#(0) ARGF9
ARCON
SMOVL C00852 BC00852 V=11.7  +MOVJ EC00852
ARCOF
SMOVL C00853 BC00853 V=800.0  +MOVJ EC00853
SMOVL C00854 BC00854 V=1000.0  +MOVJ EC00854
SFTOF3D
'EndPath W4156
'Path W4157
SFTOF3D
SFTON3D P042
MOVJ C00855 BC00855 VJ=100.00  +MOVJ EC00855 VJ=100.00
SMOVL C00856 BC00856 V=800.0  +MOVJ EC00856
SMOVL C00857 BC00857 V=150.0 PL=0  +MOVJ EC00857
ARCON
SMOVL C00858 BC00858 V=11.7  +MOVJ EC00858
ARCOF
SMOVL C00859 BC00859 V=800.0  +MOVJ EC00859
SMOVL C00860 BC00860 V=1000.0  +MOVJ EC00860
SFTOF3D
'EndPath W4157
'3
MOVJ C00861 BC00861 VJ=100.00  +MOVJ EC00861 VJ=100.00
MOVJ C00862 BC00862 VJ=100.00  +MOVJ EC00862 VJ=100.00
MOVJ C00863 BC00863 VJ=100.00  +MOVJ EC00863 VJ=100.00
MOVJ C00864 BC00864 VJ=100.00  +MOVJ EC00864 VJ=100.00
'Path W4158
SFTOF3D
SFTON3D P047
MOVJ C00865 BC00865 VJ=100.00  +MOVJ EC00865 VJ=100.00
SMOVL C00866 BC00866 V=800.0  +MOVJ EC00866
SMOVL C00867 BC00867 V=150.0 PL=0  +MOVJ EC00867
ARCON
SMOVL C00868 BC00868 V=11.7  +MOVJ EC00868
ARCOF
SMOVL C00869 BC00869 V=800.0  +MOVJ EC00869
SMOVL C00870 BC00870 V=1000.0  +MOVJ EC00870
SFTOF3D
'EndPath W4158
'Path W4159
SFTOF3D
SFTON3D P047
MOVJ C00871 BC00871 VJ=100.00  +MOVJ EC00871 VJ=100.00
SMOVL C00872 BC00872 V=800.0  +MOVJ EC00872
SMOVL C00873 BC00873 V=150.0 PL=0  +MOVJ EC00873
ARCON
SMOVL C00874 BC00874 V=11.7  +MOVJ EC00874
ARCOF
SMOVL C00875 BC00875 V=800.0  +MOVJ EC00875
SMOVL C00876 BC00876 V=1000.0  +MOVJ EC00876
SFTOF3D
'EndPath W4159
MOVJ C00877 BC00877 VJ=100.00  +MOVJ EC00877 VJ=100.00
MOVJ C00878 BC00878 VJ=100.00  +MOVJ EC00878 VJ=100.00
MOVJ C00879 BC00879 VJ=100.00  +MOVJ EC00879 VJ=100.00
MOVJ C00880 BC00880 VJ=100.00  +MOVJ EC00880 VJ=100.00
'Path W4160
SFTOF3D
SFTON3D P043
MOVJ C00881 BC00881 VJ=100.00  +MOVJ EC00881 VJ=100.00
SMOVL C00882 BC00882 V=800.0  +MOVJ EC00882
SMOVL C00883 BC00883 V=150.0 PL=0  +MOVJ EC00883
ARCON
SMOVL C00884 BC00884 V=11.7  +MOVJ EC00884
ARCOF
SMOVL C00885 BC00885 V=800.0  +MOVJ EC00885
SMOVL C00886 BC00886 V=1000.0  +MOVJ EC00886
SFTOF3D
'EndPath W4160
'Path W4161
SFTOF3D
SFTON3D P042
MOVJ C00887 BC00887 VJ=100.00  +MOVJ EC00887 VJ=100.00
SMOVL C00888 BC00888 V=800.0  +MOVJ EC00888
SMOVL C00889 BC00889 V=166.7 PL=0  +MOVJ EC00889
ARCON
SMOVL C00890 BC00890 V=11.7  +MOVJ EC00890
ARCOF
SMOVL C00891 BC00891 V=800.0  +MOVJ EC00891
SMOVL C00892 BC00892 V=1000.0  +MOVJ EC00892
SFTOF3D
'EndPath W4161
MOVJ C00893 BC00893 VJ=100.00  +MOVJ EC00893 VJ=100.00
'Path W4162
SFTOF3D
SFTON3D P046
MOVJ C00894 BC00894 VJ=100.00  +MOVJ EC00894 VJ=100.00
SMOVL C00895 BC00895 V=800.0  +MOVJ EC00895
SMOVL C00896 BC00896 V=166.7 PL=0  +MOVJ EC00896
MACRO1 MJ#(0) ARGF14
ARCON
SMOVL C00897 BC00897 V=10.0  +MOVJ EC00897
ARCOF
SMOVL C00898 BC00898 V=800.0  +MOVJ EC00898
SMOVL C00899 BC00899 V=1000.0  +MOVJ EC00899
SFTOF3D
'EndPath W4162
'Path W4163
SFTOF3D
SFTON3D P044
MOVJ C00900 BC00900 VJ=100.00  +MOVJ EC00900 VJ=100.00
SMOVL C00901 BC00901 V=800.0  +MOVJ EC00901
SMOVL C00902 BC00902 V=150.0 PL=0  +MOVJ EC00902
MACRO1 MJ#(0) ARGF9
ARCON
SMOVL C00903 BC00903 V=11.7  +MOVJ EC00903
ARCOF
SMOVL C00904 BC00904 V=800.0  +MOVJ EC00904
SMOVL C00905 BC00905 V=1000.0  +MOVJ EC00905
SFTOF3D
'EndPath W4163
MOVJ C00906 BC00906 VJ=100.00  +MOVJ EC00906 VJ=100.00
'Path W4164
SFTOF3D
SFTON3D P041
MOVJ C00907 BC00907 VJ=100.00  +MOVJ EC00907 VJ=100.00
SMOVL C00908 BC00908 V=800.0  +MOVJ EC00908
SMOVL C00909 BC00909 V=150.0 PL=0  +MOVJ EC00909
MACRO1 MJ#(0) ARGF14
ARCON
SMOVL C00910 BC00910 V=10.0  +MOVJ EC00910
SMOVL C00911 BC00911 V=10.0  +MOVJ EC00911
SMOVL C00912 BC00912 V=10.0  +MOVJ EC00912
ARCOF
SMOVL C00913 BC00913 V=800.0  +MOVJ EC00913
SMOVL C00914 BC00914 V=1000.0  +MOVJ EC00914
SFTOF3D
'EndPath W4164
JUMP *L_1
'Path W4165
SFTOF3D
SFTON3D P041
MOVJ C00915 BC00915 VJ=100.00  +MOVJ EC00915 VJ=100.00
SMOVL C00916 BC00916 V=800.0  +MOVJ EC00916
SMOVL C00917 BC00917 V=150.0 PL=0  +MOVJ EC00917
SMOVL C00918 BC00918 V=10.0  +MOVJ EC00918
ARCOF
SMOVL C00919 BC00919 V=800.0  +MOVJ EC00919
SMOVL C00920 BC00920 V=1000.0  +MOVJ EC00920
SFTOF3D
'EndPath W4165
MOVJ C00921 BC00921 VJ=100.00  +MOVJ EC00921 VJ=100.00
'Path W4166
SFTOF3D
SFTON3D P041
MOVJ C00922 BC00922 VJ=100.00  +MOVJ EC00922 VJ=100.00
SMOVL C00923 BC00923 V=800.0  +MOVJ EC00923
SMOVL C00924 BC00924 V=150.0 PL=0  +MOVJ EC00924
SMOVL C00925 BC00925 V=10.0  +MOVJ EC00925
ARCOF
SMOVL C00926 BC00926 V=800.0  +MOVJ EC00926
SMOVL C00927 BC00927 V=1000.0  +MOVJ EC00927
SFTOF3D
'EndPath W4166
*L_1
MOVJ C00928 BC00928 VJ=100.00  +MOVJ EC00928 VJ=100.00
MOVJ C00929 BC00929 VJ=100.00  +MOVJ EC00929 VJ=100.00
MOVJ C00930 BC00930 VJ=100.00  +MOVJ EC00930 VJ=100.00
END
